Staubli VAL3: OnF4.pgx

program OnF4()
  local string l_sProperty[2]
  local string l_sItem
begin
//  //调用tool or frame library
//  l_sProperty[0]="工具"
//  l_sProperty[1]="坐标系"
//  call user:SetProerty("",26,9,6,2,l_sProperty,l_sItem)
//  if l_sItem=="工具"
//    call Tool:setTool(prd:sToolName)
//    call Tool:Main(1)
//    call Tool:getTool(prd:sToolName)
//  elseIf l_sItem=="坐标系"
//    call Frame:SetFrame(prd:sFrameName)
//    call Frame:Main(1)
//    call Frame:getFrame(prd:sFrameName)
//  endIf
//  bUserRefresh=bListRefresh=true
end
